(* Logix 5000 project; controller Lab1 vendor 1 type 14 code 155 rev 20.12; software revision 20.01 *)

TASK MainTask (continuous, watchdog 500 ms) : MainProgram

MODULES
   Local : vendor 1 type 14 code 155 (PointIO 0, rev 20.12)
      A_In : 1734-IE2V (PointIO 2, rev 3.1, Input RPI 80 ms)
      Stepper_1 : vendor 10 type 150 code 185 (PointIO 5, rev 1.1, Output RPI 50 ms)
      Stepper_2 : vendor 10 type 150 code 185 (PointIO 6, rev 1.1, Output RPI 50 ms)
      Discrete_IO : Embedded (PointIO 1, rev 20.11, Output RPI 20 ms)
      A_Out : 1734-OE2V (PointIO 3, rev 3.1, Output RPI 80 ms)
      HSC : vendor 1 type 109 code 13 (PointIO 4, rev 3.1, Output RPI 80 ms)
END_MODULES

PROGRAM MainProgram   (* main routine MainRoutine *)
VAR
   STATE : INT;
   Timer_1 : TIMER := (PRE := 1000);
   Timer_2 : TIMER := (PRE := 1000);
END_VAR

ROUTINE MainRoutine   (* ladder *)
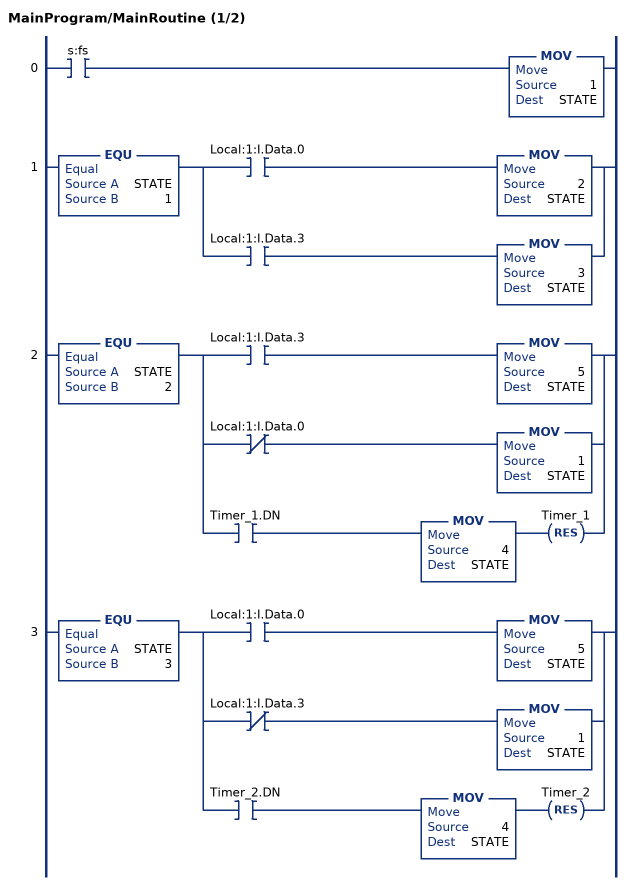
   0: XIC(s:fs)MOV(1,STATE);
   1: EQU(STATE,1)[XIC(Local:1:I.Data.0) MOV(2,STATE) ,XIC(Local:1:I.Data.3) MOV(3,STATE) ];
   2: EQU(STATE,2)[[XIC(Local:1:I.Data.3) MOV(5,STATE) ,XIO(Local:1:I.Data.0) MOV(1,STATE) ] ,XIC(Timer_1.DN) MOV(4,STATE) RES(Timer_1) ];
   3: EQU(STATE,3)[[XIC(Local:1:I.Data.0) MOV(5,STATE) ,XIO(Local:1:I.Data.3) MOV(1,STATE) ] ,XIC(Timer_2.DN) MOV(4,STATE) RES(Timer_2) ];
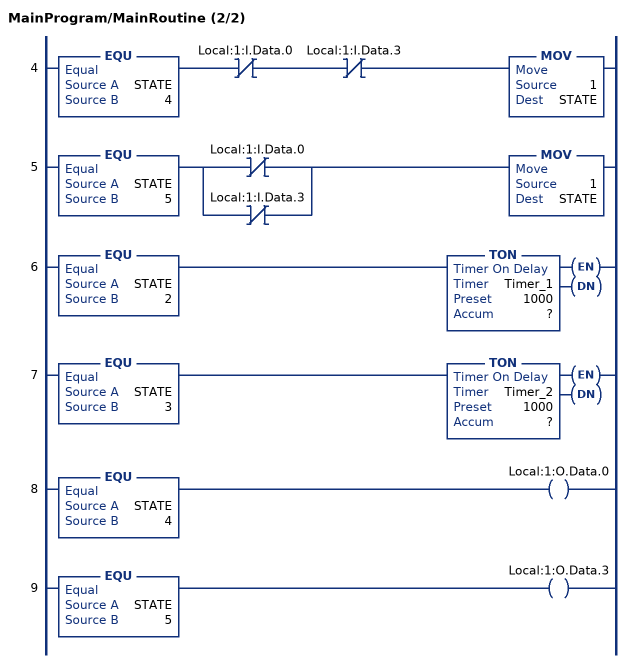
   4: EQU(STATE,4)XIO(Local:1:I.Data.0)XIO(Local:1:I.Data.3)MOV(1,STATE);
   5: EQU(STATE,5)[XIO(Local:1:I.Data.0) ,XIO(Local:1:I.Data.3) ]MOV(1,STATE);
   6: EQU(STATE,2)TON(Timer_1,?,?);
   7: EQU(STATE,3)TON(Timer_2,?,?);
   8: EQU(STATE,4)OTE(Local:1:O.Data.0);
   9: EQU(STATE,5)OTE(Local:1:O.Data.3);
END_ROUTINE
END_PROGRAM
